// Mitsubishi GX Works2 project: z12   PLC: Q02/Q02H

PROGRAM MAIN
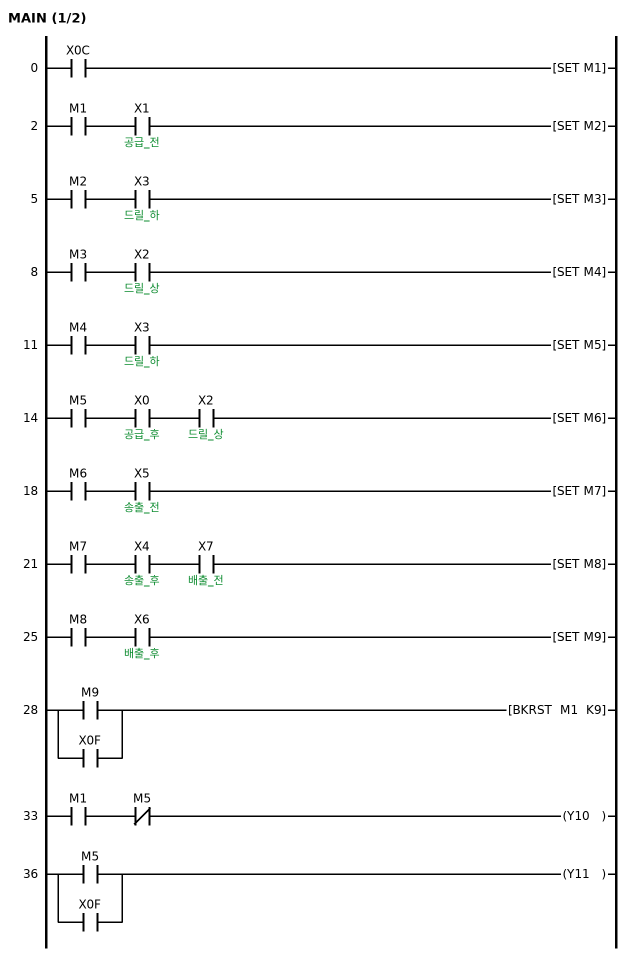
0     LD      X0C
      SET     M1
2     LD      M1
      AND     X1  ; 공급_전
      SET     M2
5     LD      M2
      AND     X3  ; 드릴_하
      SET     M3
8     LD      M3
      AND     X2  ; 드릴_상
      SET     M4
11    LD      M4
      AND     X3  ; 드릴_하
      SET     M5
14    LD      M5
      AND     X0  ; 공급_후
      AND     X2  ; 드릴_상
      SET     M6
18    LD      M6
      AND     X5  ; 송출_전
      SET     M7
21    LD      M7
      AND     X4  ; 송출_후
      AND     X7  ; 배출_전
      SET     M8
25    LD      M8
      AND     X6  ; 배출_후
      SET     M9
28    LD      M9
      OR      X0F
      BKRST   M1 K9
33    LD      M1
      ANI     M5
      OUT     Y10
36    LD      M5
      OR      X0F
      OUT     Y11
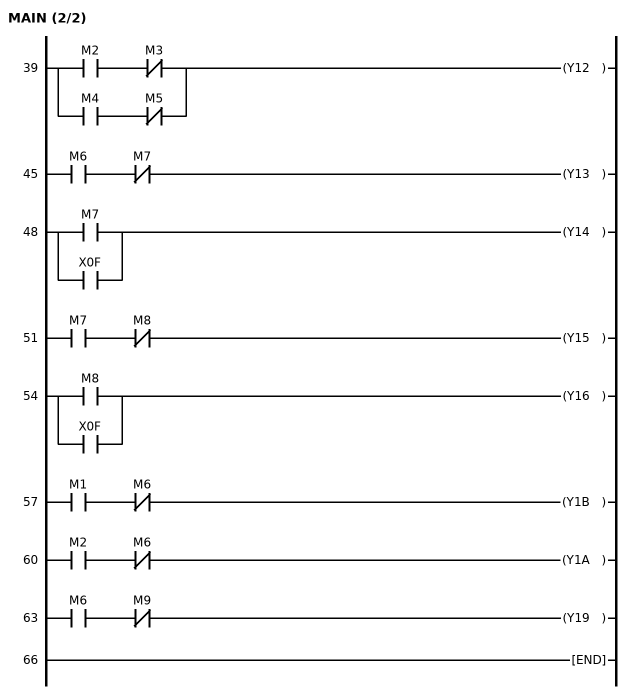
39    LD      M2
      ANI     M3
      LD      M4
      ANI     M5
      ORB
      OUT     Y12
45    LD      M6
      ANI     M7
      OUT     Y13
48    LD      M7
      OR      X0F
      OUT     Y14
51    LD      M7
      ANI     M8
      OUT     Y15
54    LD      M8
      OR      X0F
      OUT     Y16
57    LD      M1
      ANI     M6
      OUT     Y1B
60    LD      M2
      ANI     M6
      OUT     Y1A
63    LD      M6
      ANI     M9
      OUT     Y19
66    END
END_PROGRAM

// device comments not shown above
Y20  ; 공급_전
Y21  ; 공급_후
Y22  ; 드릴_하
Y23  ; 송출_전
Y24  ; 송출_후
Y25  ; 배출_전
Y26  ; 배출_후
Y29  ; RL
Y2A  ; YL
Y2B  ; GL
